FUNCTION_BLOCK Crane_MoveToStamp EXTENDS Crane_MoveBase
VAR_INPUT
END_VAR
VAR_OUTPUT
END_VAR
VAR
	// Crane_CylinderRetracted
	m_precondition: ComparisonExpression(EProcessVariables.Crane_CylinderRetracted, EComparisonType.equals, EDataType.binary, TRUE, 0, '', TRUE);
	
	// EProcessVariables.Crane_AtStamp = TRUE
	m_postcondition: ComparisonExpression(EProcessVariables.Crane_AtStamp, EComparisonType.equals, EDataType.binary, TRUE, 0, '', TRUE);
END_VAR

SUPER^();

PROPERTY AtTarget : BOOL
GET
AtTarget := m_ptrCrane^.AtStamp;
END_GET
END_PROPERTY

METHOD FB_init : BOOL
VAR_INPUT
	bInitRetains : BOOL; // if TRUE, the retain variables are initialized (warm start / cold start)
	bInCopyCode : BOOL;  // if TRUE, the instance afterwards gets moved into the copy code (online change)
		
	i_ptrCrane: POINTER TO Crane;
END_VAR
m_ptrCrane := i_ptrCrane;

m_id := EPrimitives.Crane_MoveToStamp;
m_timeout := T#30S;

Precondition := m_precondition;
Postcondition := m_postcondition;
END_METHOD

PROPERTY TargetAngle : UINT
GET
TargetAngle := 180;
END_GET
END_PROPERTY

END_FUNCTION_BLOCK

(* stored: Version 1.1.0.1
   POU Crane_MoveToStamp: Id {603c84dd-7da8-411f-b8c6-adc394ee5499}, SpecialFunc None
   Property AtTarget: Id {cdb77f6f-d5d0-4e7f-a322-2f53878bb46f}
   Get Get: Id {f1aa69a1-e7a5-4b09-9a03-f82552d62d19}
   Method FB_init: Id {e24505c1-da34-445e-be96-5791ccb9b197}
   Property TargetAngle: Id {8f3aae04-3e20-4b46-b6a3-ec6994978800}
   Get Get: Id {7145177b-79ea-425b-97f0-1d51772a8828} *)
